// TIA Portal V16 export
// export: Created 2024-03-28T09:54:30.7358906Z, ExportSetting WithDefaults, DisplayName Totally Integrated Automation Portal, DisplayVersion V16, DisplayName TIA Portal Version Control Interface, DisplayVersion V16, DisplayName TIA Portal Openness, DisplayVersion V16, DisplayName STEP 7 Professional, DisplayVersion V16, DisplayName STEP 7 Safety, DisplayVersion V16, DisplayName WinCC Advanced, DisplayVersion V16
TYPE "UR_3_T2O_Joints"
// stored: IsFailsafeCompliant false
   STRUCT
      "Joint position [rad]" : Array[0..5] of Real;
      "Joint velocity [rad/s]" : Array[0..5] of Real;
      "Joint current [A]" : Array[0..5] of Real;
      "Joint temperature [°C]" : Array[0..5] of Real;
      "Joint mode" : Array[0..5] of USInt;
      Reserved_9 { ExternalAccessible := 'False'; ExternalVisible := 'False'; ExternalWritable := 'False'} : UInt;
   END_STRUCT;
END_TYPE
